{attribute 'qualified_only'}
VAR_GLOBAL CONSTANT
	MAX_DOMAIN : UDINT := 100;
END_VAR

(* stored: Version 1.1.0.1
   GVL Param: Id {c531fecb-0b6a-43d9-880a-7990a47060a7}, ParameterList True *)
